TYPE T_Generic : __SYSTEM.AnyType; END_TYPE

(* stored: Version 1.1.0.1, ProductVersion 3.1.4024.4
   DUT T_Generic: Id {f3a06048-16d3-4fa8-98a9-33dafd9dba28} *)
